FUNCTION_BLOCK Oscillatore

VAR_INPUT
	enable : BOOL;
	t_high : TIME;
	t_low  : TIME;
END_VAR

VAR_OUTPUT
	q      : BOOL;
END_VAR

VAR
	t1     : TON();
	t2     : TON();
END_VAR

t1(in := enable, );

END_FUNCTION_BLOCK

(* stored: Version 1.1.0.1, ProductVersion 3.1.4024.12
   POU Oscillatore: Id {8ebba2c8-e785-4018-9964-69fd89c92b7c}, SpecialFunc None *)
